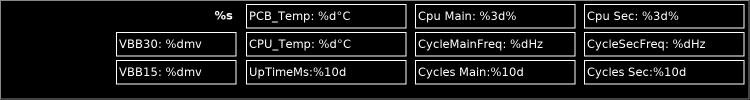
VISUALIZATION PLC_Status_Info  // 750x100
VAR_IN_OUT
	PlcStatus: SLL_IFM_CRXXXX.IFM_CRXXXX_System_STRUCT;
	Node: NodeComFB;
END_VAR
    Rectangle (246,32 160x24), "CPU_Temp: %d°C", text variable: PlcStatus.CPU_Temp
    Rectangle (415,60 160x24), "Cycles Main:%10d", text variable: PlcStatus.CycleCounter
    Rectangle (415,32 160x24), "CycleMainFreq: %dHz", text variable: PlcStatus.CycleFreq
    Rectangle (246,4 160x24), "PCB_Temp: %d°C", text variable: PlcStatus.PCB_Temp
    Rectangle (246,60 160x24), "UpTimeMs:%10d", text variable: PlcStatus.UpTimeMs
    Rectangle (116,32 120x24), "VBB30: %dmv", text variable: PlcStatus.VBB30_mV
    Rectangle (116,60 120x24), "VBB15: %dmv", text variable: PlcStatus.VBB15_mV
    Rectangle (71,4 165x23), "%s", text variable: Node.Full_Name
    Rectangle (584,4 160x24), "Cpu Sec: %3d%", text variable: TO_INT(PlcStatus.TaskInfo.fSecTaskCpuLoad)
    Rectangle (415,4 160x24), "Cpu Main: %3d%", text variable: TO_INT(PlcStatus.TaskInfo.fMainTaskCpuLoad)
    Rectangle (584,60 160x24), "Cycles Sec:%10d", text variable: PlcStatus.CycleSecCounter
    Rectangle (584,32 160x24), "CycleSecFreq: %dHz", text variable: PlcStatus.CycleSecFreq
END_VISUALIZATION

// Device/Application/LIBS/IO Diagnostics/IO Page Templates/PLC_Version_Info/PLC_Version_Info
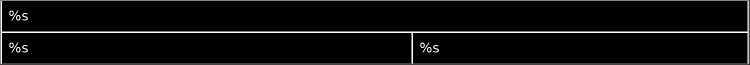
VISUALIZATION PLC_Version_Info  // 750x65
VAR_IN_OUT
	PlcVersion: PLC_Version_Unpack_FB;
END_VAR
    Textfield (1,0 747x32), "%s", text variable: PlcVersion.oMachine
    Textfield (1,32 411x32), "%s", text variable: PlcVersion.oVersion
    Textfield (412,32 336x32), "%s", text variable: PlcVersion.oCompiler
END_VISUALIZATION

// Device/Application/LIBS/IO Diagnostics/IO Page Objects/Output_Force
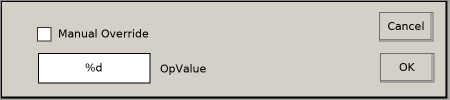
VISUALIZATION Output_Force  // 450x100
VAR_IN_OUT
	pOutputState: CRXXXX_OUTPUT_STATE_DATA;		
END_VAR
VAR
	flags: DWORD;
END_VAR
    Rectangle (0,0 447x98)
    Button (379,12 54x29), "Cancel"
        OnMouseClick:  Dialog=Current Dialog, Result=Cancel, NumpadKeypadSet=True
        OnMouseClick: execute { pOutputState.xManAuto:=0; }
    Button (380,53 54x29), "OK"
        OnMouseClick:  Dialog=Current Dialog, Result=OK, NumpadKeypadSet=True
    Checkbox (35,19 131x30), "Manual Override", variable: pOutputState.xManAuto
    Label (157,54 56x30), "OpValue"
    Rectangle (38,53 112x30), "%d", text variable: pOutputState.uiManValue
        OnMouseClick: write the text variable via VisuDialogs_Template.Numpad, min 0, max 5000, title 'Manual Value'
END_VISUALIZATION

// Device/Application/LIBS/IO Diagnostics/IO Page Objects/Output_IFM_PLC_CRXXXX_TITLE
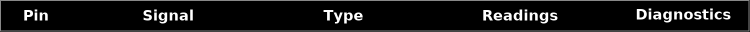
VISUALIZATION Output_IFM_PLC_CRXXXX_TITLE  // 750x32
    Textfield (398,3 244x25), "Readings"
    Textfield (629,2 109x25), "Diagnostics"
    Textfield (85,3 167x25), "Signal"
    Textfield (1,3 70x25), "Pin"
    Textfield (317,3 53x25), "Type"
END_VISUALIZATION

// Device/Application/LIBS/IO Diagnostics/IO Page Objects/Output_IFM_PLC_CRXXXX
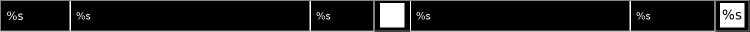
VISUALIZATION Output_IFM_PLC_CRXXXX  // 750x32
VAR_IN_OUT
	Output: CRXXXX_Output_Display;
END_VAR
VAR
END_VAR
    Textfield (410,0 220x32), "%s", text variable: Output.oMainString
        p55702900: Output.oMainStringColour
    Textfield (630,0 85x32), "%s", text variable: Output.oDiagStr
        p55702900: Output.oMainStringColour
    Textfield (70,0 240x32), "%s", text variable: Output.oSignalNameStr
    Textfield (0,0 70x32), "%s", text variable: Output.oPinDetailsStr
    Rectangle (380,3 24x24), invisible if: NOT Output.oShowDigRect, colour variable: Output.oDigRectColour
        p3450524324: Output.oDigRectColour
    Textfield (310,0 64x32), "%s", text variable: Output.oTypeStr
    Rectangle (720,3 24x24), "%s", text variable: Output.oForceText, invisible if: HMI_IO.Outputs_EnableAutoMan=0 OR Output.DisableMan=1, input disabled if: NOT HMI_IO.Outputs_EnableAutoMan OR GVL_System.HMI_OP_FORCE_DISABLE, colour variable: Output.oForceColour
        p3450524324: Output.oForceColour
        OnMouseClick:  Dialog=Output_Force, Parameters={flags: , pOutputState: Output.OpREF.OUTPUT_STATE_DATA}, Selected={1: , 0: }, OpenModal=True, OpenCentered=True
END_VISUALIZATION

// Device/Application/LIBS/IO Diagnostics/IO Page Objects/Input_IFM_PLC_CRXXXX
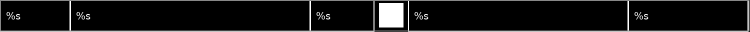
VISUALIZATION Input_IFM_PLC_CRXXXX  // 750x32
VAR_IN_OUT
	Input: CRXXXX_Input_Display;
END_VAR
VAR
END_VAR
    Textfield (408,0 220x32), "%s", text variable: Input.oMainString
        p55702900: Input.oMainStringColour
    Textfield (628,0 120x32), "%s", text variable: Input.oDiagStr
        p55702900: Input.oMainStringColour
    Textfield (70,0 240x32), "%s", text variable: Input.oSignalNameStr
    Textfield (0,0 70x32), "%s", text variable: Input.oPinDetailsStr
    Rectangle (379,3 24x24), invisible if: NOT Input.oShowDigRect, colour variable: Input.oDigRectColour
        p3450524324: Input.oDigRectColour
    Textfield (310,0 64x32), "%s", text variable: Input.oTypeStr
END_VISUALIZATION

// Device/Application/LIBS/IO Diagnostics/IO Page Objects/Input_IFM_PLC_CRXXXX_TITLE
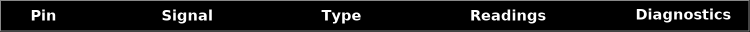
VISUALIZATION Input_IFM_PLC_CRXXXX_TITLE  // 750x32
    Textfield (386,3 244x25), "Readings"
    Textfield (629,2 109x25), "Diagnostics"
    Textfield (104,3 167x25), "Signal"
    Textfield (-1,3 89x25), "Pin"
    Textfield (315,3 53x25), "Type"
END_VISUALIZATION

// Device/Application/LIBS/IO Diagnostics/IO Page Objects/Output_Group_IFM_PLC_CRXXXX
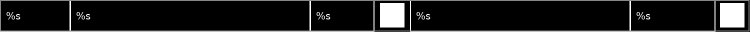
VISUALIZATION Output_Group_IFM_PLC_CRXXXX  // 750x32
{attribute 'VAR_IN_OUT_AS_POINTER'}
VAR_IN_OUT
	Output: CRXXXX_Output_Group_Display;
END_VAR
VAR
END_VAR
    Textfield (410,0 220x32), "%s", text variable: Output.oMainString
        p55702900: Output.oMainStringColour
    Textfield (630,0 85x32), "%s", text variable: Output.oDiagStr
        p55702900: Output.oMainStringColour
    Textfield (70,0 240x32), "%s", text variable: Output.oSignalNameStr
    Textfield (0,0 70x32), "%s", text variable: Output.oPinDetailsStr
    Rectangle (380,3 24x24), invisible if: NOT Output.oShowDigRect, colour variable: Output.oDigRectColour
        p3450524324: Output.oDigRectColour
    Textfield (310,0 64x32), "%s", text variable: Output.oTypeStr
    Rectangle (720,3 24x24), invisible if: NOT HMI_IO.Outputs_EnableAutoMan, input disabled if: NOT HMI_IO.Outputs_EnableAutoMan OR GVL_System.HMI_OP_FORCE_DISABLE
        OnMouseClick:  Dialog=Output_Force, Parameters={flags: , pOutputState: Output.OpGrpREF.OUTPUT_STATE_DATA}, Selected={1: , 0: }, OpenModal=True, OpenCentered=True
END_VISUALIZATION

// Device/Application/LIBS/IO Diagnostics/IO Page Templates/CR0709/Visualization_CR0709_Op_G0
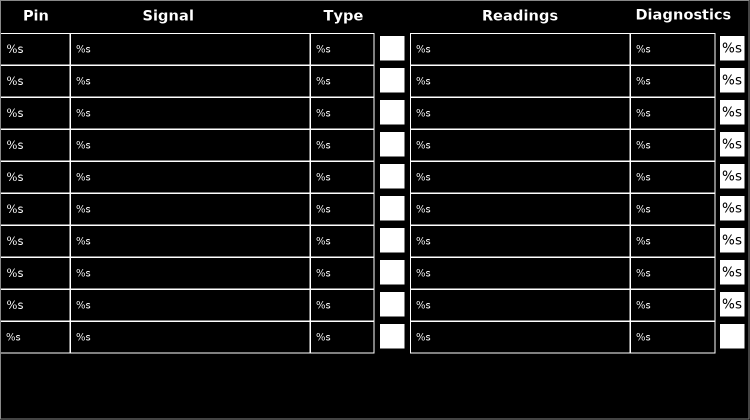
VISUALIZATION Visualization_CR0709_Op_G0  // 750x420
VAR_IN_OUT
	HMI_PLC_IO: HMI_PLC_CR0709_IO;
END_VAR
    Frame (0,33 800x32)
        shows Output_IFM_PLC_CRXXXX(Output := HMI_PLC_IO.OUT0000)
    Frame (0,0 800x32)
        shows Output_IFM_PLC_CRXXXX_TITLE()
    Frame (0,65 762x32)
        shows Output_IFM_PLC_CRXXXX(Output := HMI_PLC_IO.OUT0001)
    Frame (0,97 762x32)
        shows Output_IFM_PLC_CRXXXX(Output := HMI_PLC_IO.OUT0002)
    Frame (0,129 762x32)
        shows Output_IFM_PLC_CRXXXX(Output := HMI_PLC_IO.OUT0003)
    Frame (0,161 762x32)
        shows Output_IFM_PLC_CRXXXX(Output := HMI_PLC_IO.OUT0004)
    Frame (0,193 762x32)
        shows Output_IFM_PLC_CRXXXX(Output := HMI_PLC_IO.OUT0005)
    Frame (0,225 762x32)
        shows Output_IFM_PLC_CRXXXX(Output := HMI_PLC_IO.OUT0006)
    Frame (0,257 762x32)
        shows Output_IFM_PLC_CRXXXX(Output := HMI_PLC_IO.OUT0007)
    Frame (0,289 762x32)
        shows Output_IFM_PLC_CRXXXX(Output := HMI_PLC_IO.OUT0008)
    Frame (0,321 780x32)
        shows Output_Group_IFM_PLC_CRXXXX(Output := HMI_PLC_IO.GROUP0)
END_VISUALIZATION

// Device/Application/LIBS/IO Diagnostics/IO Page Templates/CR0709/Visualization_CR0709_Op_G2
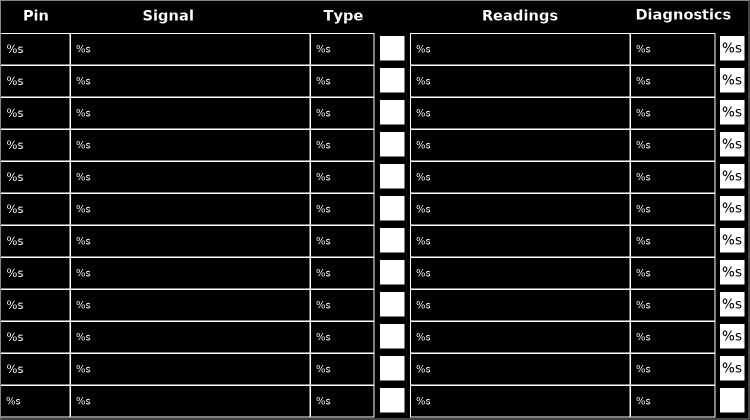
VISUALIZATION Visualization_CR0709_Op_G2  // 750x420
VAR_IN_OUT
	HMI_PLC_IO: HMI_PLC_CR0709_IO;
END_VAR
    Frame (0,33 762x32)
        shows Output_IFM_PLC_CRXXXX(Output := HMI_PLC_IO.OUT0200)
    Frame (0,0 800x32)
        shows Output_IFM_PLC_CRXXXX_TITLE()
    Frame (0,65 762x32)
        shows Output_IFM_PLC_CRXXXX(Output := HMI_PLC_IO.OUT0201)
    Frame (0,97 762x32)
        shows Output_IFM_PLC_CRXXXX(Output := HMI_PLC_IO.OUT0202)
    Frame (0,129 762x32)
        shows Output_IFM_PLC_CRXXXX(Output := HMI_PLC_IO.OUT0203)
    Frame (0,161 762x32)
        shows Output_IFM_PLC_CRXXXX(Output := HMI_PLC_IO.OUT0204)
    Frame (0,193 762x32)
        shows Output_IFM_PLC_CRXXXX(Output := HMI_PLC_IO.OUT0205)
    Frame (0,225 762x32)
        shows Output_IFM_PLC_CRXXXX(Output := HMI_PLC_IO.OUT0206)
    Frame (0,257 762x32)
        shows Output_IFM_PLC_CRXXXX(Output := HMI_PLC_IO.OUT0207)
    Frame (0,289 762x32)
        shows Output_IFM_PLC_CRXXXX(Output := HMI_PLC_IO.OUT0208)
    Frame (0,385 780x32)
        shows Output_Group_IFM_PLC_CRXXXX(Output := HMI_PLC_IO.GROUP2)
    Frame (0,321 762x32)
        shows Output_IFM_PLC_CRXXXX(Output := HMI_PLC_IO.OUT3000)
    Frame (0,353 762x32)
        shows Output_IFM_PLC_CRXXXX(Output := HMI_PLC_IO.OUT3001)
END_VISUALIZATION

// Device/Application/App_Common/Vizualisations/Main/Visualization_Net_Status_Adv
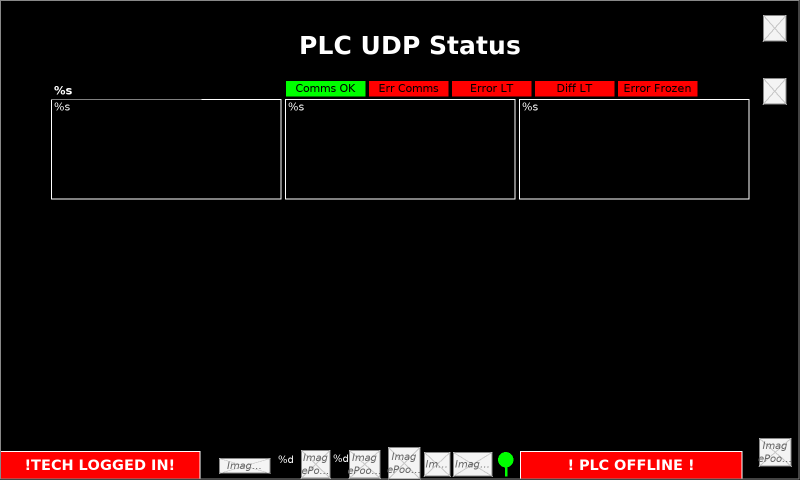
VISUALIZATION Visualization_Net_Status_Adv  // 800x480
    Frame (0,0 800x480)
        shows Visualization_Template()
    Label (219,30 382x30), "PLC UDP Status"
    Frame (50,80 700x120)
        shows PLC_UDP_Info(UDP_Info := PLC_SYSTEM.CHASSIS_UDP_Info_Viz)
    Image (763,15 23x26), invisible if: Nav.Footer_ShowNavLeft=0, image: ImagePool.Page_nav_left
    Image (763,78 23x26), invisible if: Nav.Footer_ShowNavRight=0, image: ImagePool.Page_nav_right
END_VISUALIZATION

// Device/Application/App_Common/Vizualisations/Main/Layout/Simulation/Visualization_SIM_IO
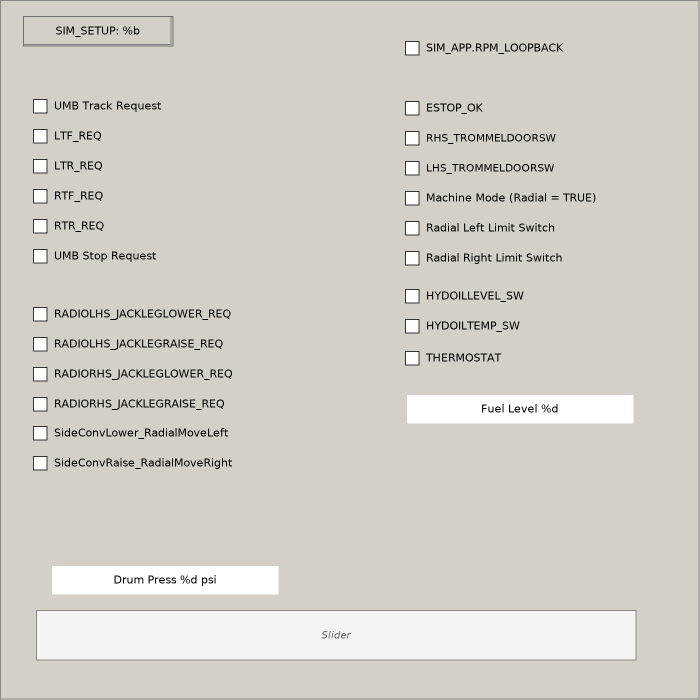
VISUALIZATION Visualization_SIM_IO  // 700x700
    Checkbox (403,33 188x30), "SIM_APP.RPM_LOOPBACK", variable: SIM_APP.RPM_LOOPBACK
    Checkbox (403,93 150x30), "ESTOP_OK", variable: Machine_IO.Inputs.ESTOP_OK.Dig
    Checkbox (403,123 150x30), "RHS_TROMMELDOORSW", variable: Machine_IO.Inputs.RHS_TROMMELDOORSW.Dig
    Checkbox (403,153 150x30), "LHS_TROMMELDOORSW", variable: Machine_IO.Inputs.LHS_TROMMELDOORSW.Dig
    Button (23,16 150x30), "SIM_SETUP: %b", text variable: SIM_APP.SIM_SETUP
        tap SIM_APP.SIM_SETUP
    Checkbox (403,183 231x30), "Machine Mode (Radial = TRUE)", variable: Machine_IO.Inputs.MachineMode.Dig
    Checkbox (403,213 250x30), "Radial Left Limit Switch", variable: Machine_IO.Inputs.Radial_LeftLimitSwitch.Dig
    Checkbox (403,243 250x30), "Radial Right Limit Switch", variable: Machine_IO.Inputs.Radial_RightLimitSwitch.Dig
    Checkbox (31,91 200x30), "UMB Track Request", variable: Machine_IO.Inputs.UMBTRACKREQ.Dig
    Checkbox (31,121 200x30), "LTF_REQ", variable: Machine_IO.Inputs.LTF_REQ.Dig
    Checkbox (31,151 200x30), "LTR_REQ", variable: Machine_IO.Inputs.LTR_REQ.Dig
    Checkbox (31,181 200x30), "RTF_REQ", variable: Machine_IO.Inputs.RTF_REQ.Dig
    Checkbox (31,211 200x30), "RTR_REQ", variable: Machine_IO.Inputs.RTR_REQ.Dig
    Checkbox (31,241 200x30), "UMB Stop Request", variable: Machine_IO.Inputs.UMBMACHINESTOP.Dig
    Slider (36,610 600x50), variable: Machine_IO.Inputs.DRUM_PRESSURE.ScaledReal, scale 0..3500
    Textfield (51,565 228x30), "Drum Press %d psi", text variable: Machine_IO.Inputs.DRUM_PRESSURE.ScaledReal
        OnMouseClick: write the text variable via Edit
    Checkbox (31,299 250x30), "RADIOLHS_JACKLEGLOWER_REQ", variable: Machine_IO.Inputs.RADIOLHS_JACKLEGLOWER_REQ.Dig
    Checkbox (31,329 250x30), "RADIOLHS_JACKLEGRAISE_REQ", variable: Machine_IO.Inputs.RADIOLHS_JACKLEGRAISE_REQ.Dig
    Checkbox (31,359 250x30), "RADIORHS_JACKLEGLOWER_REQ", variable: Machine_IO.Inputs.RADIORHS_JACKLEGLOWER_REQ.Dig
    Checkbox (31,389 250x30), "RADIORHS_JACKLEGRAISE_REQ", variable: Machine_IO.Inputs.RADIORHS_JACKLEGRAISE_REQ.Dig
    Checkbox (31,418 250x30), "SideConvLower_RadialMoveLeft", variable: Machine_IO.Inputs.SideConvLower_RadialMoveLeft.Dig
    Checkbox (31,448 250x30), "SideConvRaise_RadialMoveRight", variable: Machine_IO.Inputs.SideConvRaise_RadialMoveRight.Dig
    Checkbox (403,281 250x30), "HYDOILLEVEL_SW", variable: Machine_IO.Inputs.HYDOILLEVEL_SW.Dig
    Checkbox (403,311 250x30), "HYDOILTEMP_SW", variable: Machine_IO.Inputs.HYDOILTEMP_SW.Dig
    Checkbox (403,343 250x30), "THERMOSTAT", variable: Machine_IO.Inputs.THERMOSTAT.Dig
    Textfield (406,394 228x30), "Fuel Level %d", text variable: Machine_IO.Inputs.FUELLEVEL_PERCENT.ScaledReal
        OnMouseClick: write the text variable via Edit
END_VISUALIZATION

// Device/Application/App_Common/Vizualisations/Main/Visualization_Net_Status
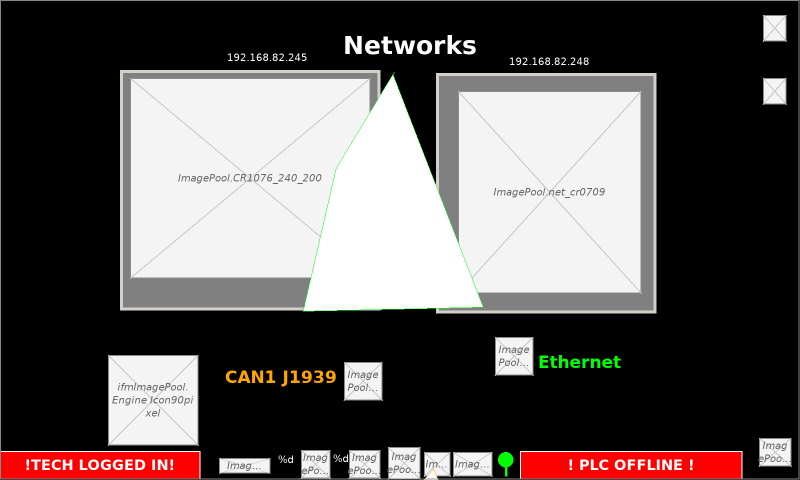
VISUALIZATION Visualization_Net_Status  // 800x480
    Frame (0,0 800x480)
        shows Visualization_Template()
    Frame (0,21 800x424)
        shows Visualization_Net_Background()
    Polygon (483,307) (303,311) (336,168) (394,72) (393,75)
    Label (190,363 150x28), "CAN1 J1939"
    Label (535,348 174x28), "Ethernet"
    Label (219,30 382x30), "Networks"
    Polygon (507,639) (389,729) (311,591) (433,470) (433,468)
    Image (495,337 38x38), invisible if: UDP_COMS_RX.CHASSIS_PLC_RED_CROSS=0, image: ImagePool.red-cross
    Image (344,362 38x38), invisible if: GVL_Engine.EngineHrs>0, image: ImagePool.red-cross
    Image (763,15 23x26), invisible if: Nav.Footer_ShowNavLeft=0, image: ImagePool.Page_nav_left
    Image (763,78 23x26), invisible if: Nav.Footer_ShowNavRight=0, image: ImagePool.Page_nav_right
    Image (108,355 90x90), image: ifmImagePool.Engine Icon90pixel
END_VISUALIZATION

// Device/Application/LIBS/IO Diagnostics/IO Page Templates/CR0709/Visualization_CR0709_Ip_G0
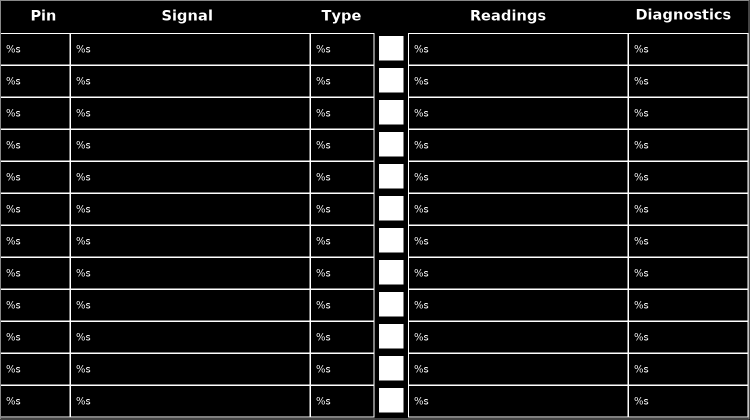
VISUALIZATION Visualization_CR0709_Ip_G0  // 750x420
VAR_IN_OUT
	HMI_PLC_IO: HMI_PLC_CR0709_IO;
END_VAR
    Frame (0,33 762x32)
        shows Input_IFM_PLC_CRXXXX(Input := HMI_PLC_IO.IN0100)
    Frame (0,0 750x32)
        shows Input_IFM_PLC_CRXXXX_TITLE()
    Frame (0,65 762x32)
        shows Input_IFM_PLC_CRXXXX(Input := HMI_PLC_IO.IN0101)
    Frame (0,97 762x32)
        shows Input_IFM_PLC_CRXXXX(Input := HMI_PLC_IO.IN0102)
    Frame (0,129 762x32)
        shows Input_IFM_PLC_CRXXXX(Input := HMI_PLC_IO.IN0103)
    Frame (0,161 762x32)
        shows Input_IFM_PLC_CRXXXX(Input := HMI_PLC_IO.IN0200)
    Frame (0,193 762x32)
        shows Input_IFM_PLC_CRXXXX(Input := HMI_PLC_IO.IN0201)
    Frame (0,225 762x32)
        shows Input_IFM_PLC_CRXXXX(Input := HMI_PLC_IO.IN0202)
    Frame (0,257 762x32)
        shows Input_IFM_PLC_CRXXXX(Input := HMI_PLC_IO.IN0203)
    Frame (0,289 762x32)
        shows Input_IFM_PLC_CRXXXX(Input := HMI_PLC_IO.IN0600)
    Frame (0,321 762x32)
        shows Input_IFM_PLC_CRXXXX(Input := HMI_PLC_IO.IN0601)
    Frame (0,353 762x32)
        shows Input_IFM_PLC_CRXXXX(Input := HMI_PLC_IO.IN0602)
    Frame (0,385 762x32)
        shows Input_IFM_PLC_CRXXXX(Input := HMI_PLC_IO.IN0603)
END_VISUALIZATION

// Device/Application/LIBS/IO Diagnostics/IO Page Templates/CR0709/Visualization_CR0709_Ip_G1
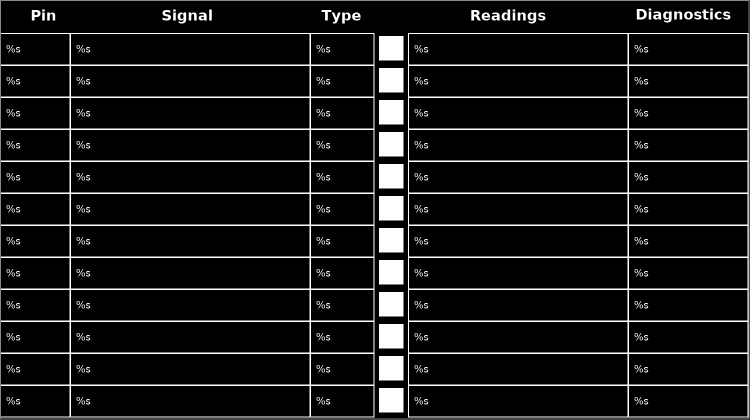
VISUALIZATION Visualization_CR0709_Ip_G1  // 750x420
VAR_IN_OUT
	HMI_PLC_IO: HMI_PLC_CR0709_IO;
END_VAR
    Frame (0,33 762x32)
        shows Input_IFM_PLC_CRXXXX(Input := HMI_PLC_IO.IN0700)
    Frame (0,0 801x32)
        shows Input_IFM_PLC_CRXXXX_TITLE()
    Frame (0,65 762x32)
        shows Input_IFM_PLC_CRXXXX(Input := HMI_PLC_IO.IN0701)
    Frame (0,97 762x32)
        shows Input_IFM_PLC_CRXXXX(Input := HMI_PLC_IO.IN0702)
    Frame (0,129 762x32)
        shows Input_IFM_PLC_CRXXXX(Input := HMI_PLC_IO.IN0703)
    Frame (0,161 762x32)
        shows Input_IFM_PLC_CRXXXX(Input := HMI_PLC_IO.IN0000)
    Frame (0,193 762x32)
        shows Input_IFM_PLC_CRXXXX(Input := HMI_PLC_IO.IN0001)
    Frame (0,225 762x32)
        shows Input_IFM_PLC_CRXXXX(Input := HMI_PLC_IO.IN0002)
    Frame (0,257 762x32)
        shows Input_IFM_PLC_CRXXXX(Input := HMI_PLC_IO.IN0003)
    Frame (0,289 762x32)
        shows Input_IFM_PLC_CRXXXX(Input := HMI_PLC_IO.IN0500)
    Frame (0,321 762x32)
        shows Input_IFM_PLC_CRXXXX(Input := HMI_PLC_IO.IN0501)
    Frame (0,353 762x32)
        shows Input_IFM_PLC_CRXXXX(Input := HMI_PLC_IO.IN0502)
    Frame (0,385 762x32)
        shows Input_IFM_PLC_CRXXXX(Input := HMI_PLC_IO.IN0503)
END_VISUALIZATION

// Device/Application/App_Common/Vizualisations/Main/Layout/Visualization_Net_Background
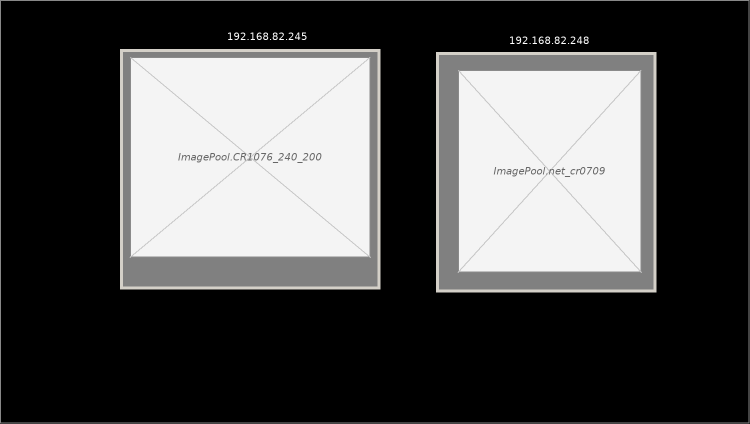
VISUALIZATION Visualization_Net_Background  // 750x424
    Rectangle (120,49 260x240)
    Rectangle (436,52 220x240)
    Image (458,70 183x202), image: ImagePool.net_cr0709
    Rectangle (501,31 97x19), "192.168.82.248"
    Rectangle (219,27 97x19), "192.168.82.245"
    Image (130,57 240x200), image: ImagePool.CR1076_240_200
END_VISUALIZATION

// Device/Application/App_Common/Vizualisations/Main/Visualization_Settings_Misc
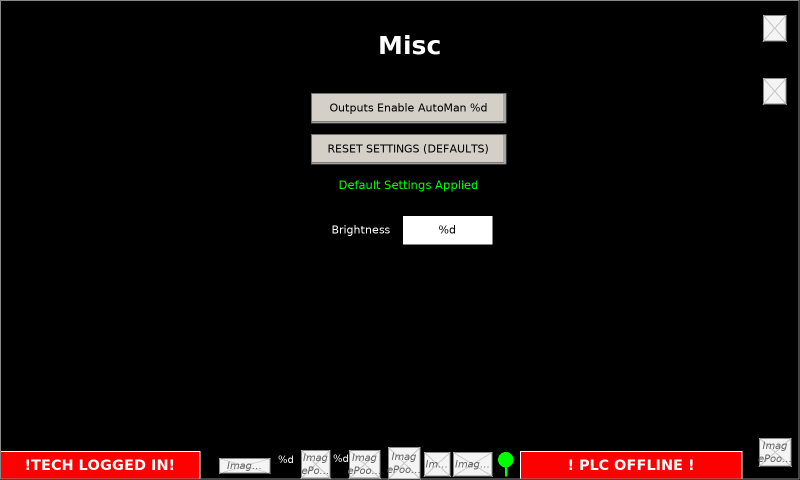
VISUALIZATION Visualization_Settings_Misc  // 800x480
    Frame (0,0 800x480)
        shows Visualization_Template()
    Label (219,30 382x30), "Misc"
    Button (311,93 195x30), "Outputs Enable AutoMan %d", text variable: HMI_IO.Outputs_EnableAutoMan, invisible if: NOT GVL_System.Access_Level_Tech
        toggle HMI_IO.Outputs_EnableAutoMan
    Label (317,215 76x30), "Brightness"
    Rectangle (402,215 91x30), "%d", text variable: GVL_Persistant.Brightness
        OnValueChanged: execute {  }
        OnValueChanged: write the text variable via Default, min LCD_Brighness_Control.Brightness_Min, max LCD_Brighness_Control.Brightness_Max
        OnMouseClick: write the text variable via VisuDialogs_Template.Numpad, min 10, max 100, title 'Brighntess %'
    Button (311,134 195x30), "RESET SETTINGS (DEFAULTS)", invisible if: GVL_System.Access_Level_Tech=0
        tap PLC_SYSTEM.Reset_Settings
    Label (311,174 195x22), "Default Settings Applied", invisible if: PLC_SYSTEM.Reset_Settings_Applied=0
    Image (763,15 23x26), invisible if: Nav.Footer_ShowNavLeft=0, image: ImagePool.Page_nav_left
    Image (763,78 23x26), invisible if: Nav.Footer_ShowNavRight=0, image: ImagePool.Page_nav_right
END_VISUALIZATION

// Device/Application/App_Common/Vizualisations/Main/Visualization_PLC_Status
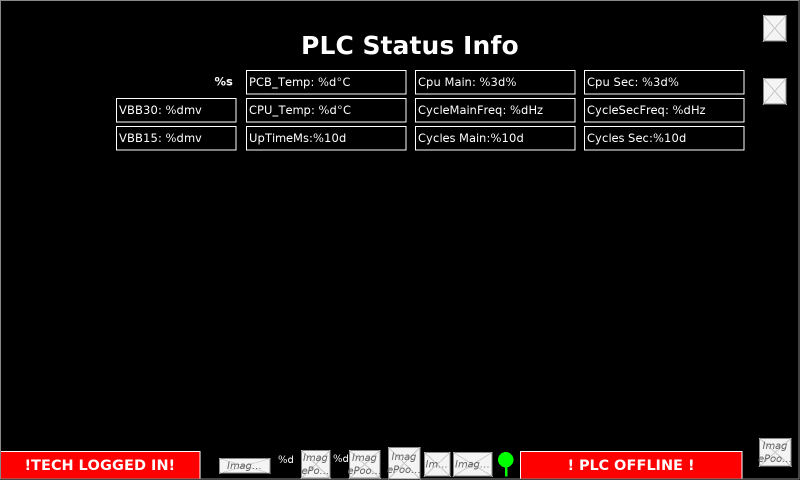
VISUALIZATION Visualization_PLC_Status  // 800x480
    Frame (0,0 800x480)
        shows Visualization_Template()
    Label (219,30 382x30), "PLC Status Info"
    Frame (0,66 800x65)
        shows PLC_Status_Info(PlcStatus := NVL_IO_CHASSIS.System, Node := Machine_IO.Node_CHASSIS)
    Image (763,15 23x26), invisible if: Nav.Footer_ShowNavLeft=0, image: ImagePool.Page_nav_left
    Image (763,78 23x26), invisible if: Nav.Footer_ShowNavRight=0, image: ImagePool.Page_nav_right
END_VISUALIZATION

// Device/Application/App_Common/Vizualisations/Main/Visualization_Settings_RTC
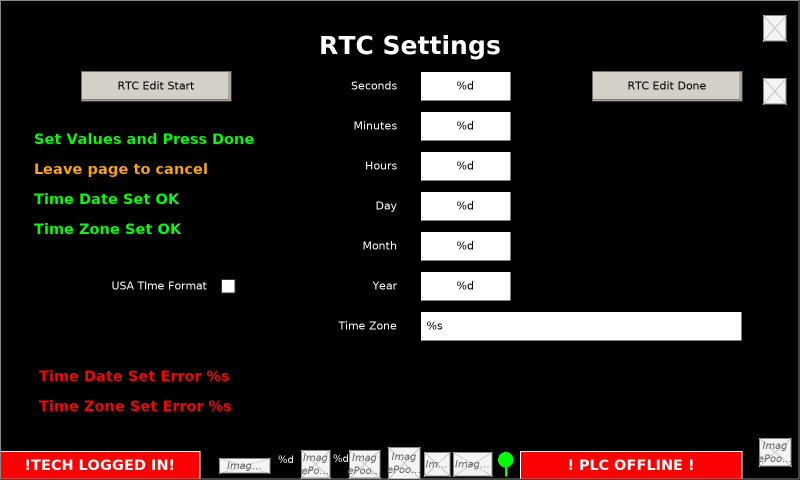
VISUALIZATION Visualization_Settings_RTC  // 800x480
    Frame (0,0 800x480)
        shows Visualization_Template()
    Label (219,30 382x30), "RTC Settings"
    Label (300,271 100x30), "Year"
    Rectangle (420,271 91x30), "%d", text variable: CR1140_RTC_Edit.RTC_Temp.uiYear, input disabled if: CR1140_RTC_Edit.RTC_Edit_Start=0
        OnValueChanged: execute { CR1140_RTC_Edit.RTC_Edit_Start:=1; }
        OnMouseClick: write the text variable via VisuDialogs_Template.Numpad, min 2000, max 3000, title 'Years in YYYYY format'
    Label (300,231 100x30), "Month"
    Rectangle (420,231 91x30), "%d", text variable: CR1140_RTC_Edit.RTC_Temp.uiMonth, input disabled if: CR1140_RTC_Edit.RTC_Edit_Start=0
        OnValueChanged: execute { CR1140_RTC_Edit.RTC_Edit_Start:=1; }
        OnMouseClick: write the text variable via VisuDialogs_Template.Numpad, min 1, max 12, title 'Month'
    Label (300,191 100x30), "Day"
    Rectangle (420,191 91x30), "%d", text variable: CR1140_RTC_Edit.RTC_Temp.uiDay, input disabled if: CR1140_RTC_Edit.RTC_Edit_Start=0
        OnValueChanged: execute { CR1140_RTC_Edit.RTC_Edit_Start:=1; }
        OnMouseClick: write the text variable via VisuDialogs_Template.Numpad, min 1, max 31, title 'Day of Month'
    Label (300,151 100x30), "Hours"
    Rectangle (420,151 91x30), "%d", text variable: CR1140_RTC_Edit.RTC_Temp.uiHour, input disabled if: CR1140_RTC_Edit.RTC_Edit_Start=0
        OnValueChanged: execute { CR1140_RTC_Edit.RTC_Edit_Start:=1; }
        OnMouseClick: write the text variable via VisuDialogs_Template.Numpad, min 0, max 23, title 'Hours (24hr)'
    Label (300,111 100x30), "Minutes"
    Rectangle (420,111 91x30), "%d", text variable: CR1140_RTC_Edit.RTC_Temp.uiMinute, input disabled if: CR1140_RTC_Edit.RTC_Edit_Start=0
        OnValueChanged: execute { CR1140_RTC_Edit.RTC_Edit_Start:=1; }
        OnMouseClick: write the text variable via VisuDialogs_Template.Numpad, min 0, max 59, title 'Minutes'
    Label (300,71 100x30), "Seconds"
    Rectangle (420,71 91x30), "%d", text variable: CR1140_RTC_Edit.RTC_Temp.uiSeconds, input disabled if: CR1140_RTC_Edit.RTC_Edit_Start=0
        OnValueChanged: execute { CR1140_RTC_Edit.RTC_Edit_Start:=1; }
        OnMouseClick: write the text variable via VisuDialogs_Template.Numpad, min 0, max 59, title 'Secondst'
    Button (81,71 150x30), "RTC Edit Start"
        toggle CR1140_RTC_Edit.RTC_Edit_Start p2164770859=TRUE
    Button (592,71 150x30), "RTC Edit Done", input disabled if: CR1140_RTC_Edit.RTC_Edit_Start=0
        tap CR1140_RTC_Edit.RTC_Edit_Done
    Label (31,124 250x30), "Set Values and Press Done", invisible if: CR1140_RTC_Edit.RTC_Edit_Start=0
    Label (31,154 250x30), "Leave page to cancel", invisible if: CR1140_RTC_Edit.RTC_Edit_Start=0
    Label (300,311 100x30), "Time Zone"
    Rectangle (420,311 322x30), "%s", text variable: CR1140_RTC_Edit.RTC_Timezone, input disabled if: CR1140_RTC_Edit.RTC_Edit_Start=0
        OnValueChanged: execute { CR1140_RTC_Edit.RTC_Edit_Start:=1; }
        OnMouseClick: write the text variable via VisuDialogs_Template.Keypad, title 'Time Zone - see docs'
    Label (31,184 250x30), "Time Date Set OK", invisible if: CR1140_RTC_Edit.TimeDateSetOK=0
    Label (31,214 250x30), "Time Zone Set OK", invisible if: CR1140_RTC_Edit.ZoneSetOK=0
    Rectangle (31,391 700x30), "Time Zone Set Error %s", text variable: CR1140_RTC_Edit.ZoneSetErrorCode, invisible if: CR1140_RTC_Edit.ZoneSetError=0
    Rectangle (31,361 700x30), "Time Date Set Error %s", text variable: CR1140_RTC_Edit.TimeDateSetErrorCode, invisible if: CR1140_RTC_Edit.TimeDateSetError=0
    Checkbox (219,271 33x30), variable: GVL_Persistant.Sys_Settings.USA_TIme_Format
    Label (94,271 116x30), "USA TIme Format"
    Image (763,15 23x26), invisible if: Nav.Footer_ShowNavLeft=0, image: ImagePool.Page_nav_left
    Image (763,78 23x26), invisible if: Nav.Footer_ShowNavRight=0, image: ImagePool.Page_nav_right
END_VISUALIZATION

// Device/Application/App_Common/Vizualisations/Main/Layout/Simulation/Visualization_SIM_IO_AUX
VISUALIZATION Visualization_SIM_IO_AUX  // 700x700
END_VISUALIZATION

// Device/Application/App_Common/Vizualisations/Main/Visualization_Settings_IO_Log
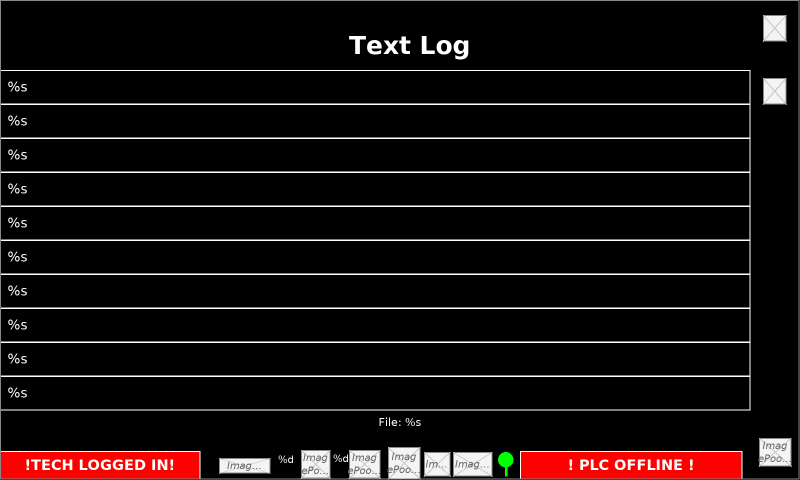
VISUALIZATION Visualization_Settings_IO_Log  // 800x480
    Frame (0,0 800x480)
        shows Visualization_Template()
    Label (219,30 382x30), "Text Log"
    Rectangle (0,70 750x34), "%s", text variable: PLC_LOGGING.LOG_LINES[0]
    Rectangle (0,104 750x34), "%s", text variable: PLC_LOGGING.LOG_LINES[1]
    Rectangle (0,138 750x34), "%s", text variable: PLC_LOGGING.LOG_LINES[2]
    Rectangle (0,172 750x34), "%s", text variable: PLC_LOGGING.LOG_LINES[3]
    Rectangle (0,206 750x34), "%s", text variable: PLC_LOGGING.LOG_LINES[4]
    Rectangle (0,240 750x34), "%s", text variable: PLC_LOGGING.LOG_LINES[5]
    Rectangle (0,274 750x34), "%s", text variable: PLC_LOGGING.LOG_LINES[6]
    Rectangle (0,308 750x34), "%s", text variable: PLC_LOGGING.LOG_LINES[7]
    Rectangle (0,342 750x34), "%s", text variable: PLC_LOGGING.LOG_LINES[8]
    Rectangle (0,376 750x34), "%s", text variable: PLC_LOGGING.LOG_LINES[9]
    Rectangle (250,410 300x25), "File: %s", text variable: GVL_Logging.Main_Log_Filename
    Image (763,15 23x26), invisible if: Nav.Footer_ShowNavLeft=0, image: ImagePool.Page_nav_left
    Image (763,78 23x26), invisible if: Nav.Footer_ShowNavRight=0, image: ImagePool.Page_nav_right
END_VISUALIZATION

// Device/Application/App_Common/Vizualisations/Main/Visualization_Settings_1
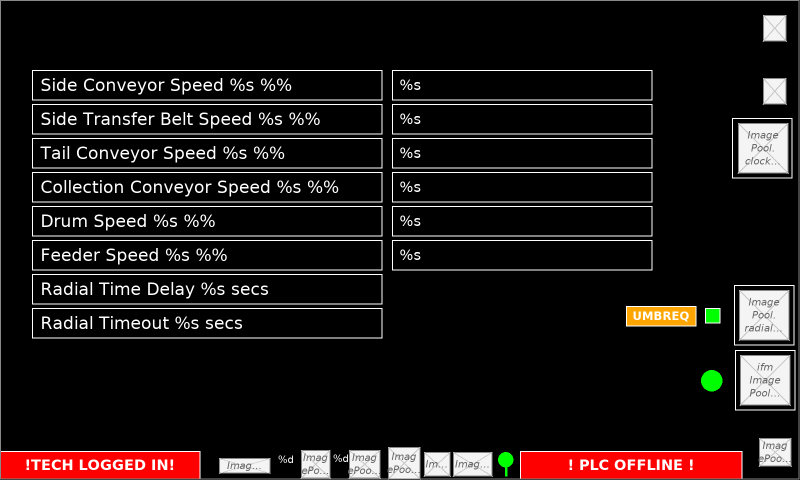
VISUALIZATION Visualization_Settings_1  // 800x480
    Frame (0,0 800x480)
        shows Visualization_Template()
    Rectangle (32,240 350x30), "Feeder Speed %s %%", text variable: GVL_Persistant.App_Settings.FeederSpd_Percent
        OnMouseClick: write the text variable via VisuDialogs_Template.Numpad, min 0, max 100, title "Feeder Speed %"
    Rectangle (32,206 350x30), "Drum Speed %s %%", text variable: GVL_Persistant.App_Settings.DrumSpd_Percent
        OnMouseClick: write the text variable via VisuDialogs_Template.Numpad, min 0, max 100, title "Drum Speed %"
    Rectangle (32,172 350x30), "Collection Conveyor Speed %s %%", text variable: GVL_Persistant.App_Settings.CollectConvSpd_Percent
        OnMouseClick: write the text variable via VisuDialogs_Template.Numpad, min 0, max 100, title "Collection Conveyor Speed %"
    Rectangle (32,70 350x30), "Stockpile Conv Speed %s %%", text variable: GVL_Persistant.App_Settings.SideConvSpd_Percent, invisible if: GVL_APP.MachineModelRadial=0
        OnMouseClick: write the text variable via VisuDialogs_Template.Numpad, min 0, max 100, title "Stockpile Conv. Speed %"
    Rectangle (32,138 350x30), "Tail Conveyor Speed %s %%", text variable: GVL_Persistant.App_Settings.TailConvSpd_Percent
        OnMouseClick: write the text variable via VisuDialogs_Template.Numpad, min 0, max 100, title "Tail Conveyor Speed %"
    Image (740,355 50x50), image: ifmImagePool.LeverValve50pixel
    Ellipse (701,370 21x21), invisible if: GVL_Machine.SetupDumpValveOn=0
    RoundedRectangle (735,350 60x60)
    Image (763,15 23x26), invisible if: Nav.Footer_ShowNavLeft=0, image: ImagePool.Page_nav_left
    Image (763,78 23x26), invisible if: Nav.Footer_ShowNavRight=0, image: ImagePool.Page_nav_right
    Rectangle (392,240 260x30), "%s", text variable: AutoManSelButtons.PWM_Op_FeederSpeed_Status_Str
        OnMouseClick: write the text variable via VisuDialogs_Template.Numpad, min 0, max 100, title "Feeder Speed %"
    Rectangle (392,206 260x30), "%s", text variable: AutoManSelButtons.PWM_Op_DrumSpeed_Status_Str
        OnMouseClick: write the text variable via VisuDialogs_Template.Numpad, min 0, max 100, title "Feeder Speed %"
    Rectangle (392,172 260x30), "%s", text variable: AutoManSelButtons.PWM_Op_CollectionConveyor_Status_Str
        OnMouseClick: write the text variable via VisuDialogs_Template.Numpad, min 0, max 100, title "Feeder Speed %"
    Rectangle (392,138 260x30), "%s", text variable: AutoManSelButtons.PWM_Op_TailConveyor_Status_Str
        OnMouseClick: write the text variable via VisuDialogs_Template.Numpad, min 0, max 100, title "Feeder Speed %"
    Rectangle (392,104 260x30), "%s", text variable: AutoManSelButtons.PWM_Op_SideTransfer_Status_Str, invisible if: GVL_APP.MachineModelRadial=1
        OnMouseClick: write the text variable via VisuDialogs_Template.Numpad, min 0, max 100, title "Feeder Speed %"
    Rectangle (392,70 260x30), "%s", text variable: AutoManSelButtons.PWM_Op_SideConveyor_Status_Str
        OnMouseClick: write the text variable via VisuDialogs_Template.Numpad, min 0, max 100, title "Feeder Speed %"
    Image (738,123 48x50), invisible if: GVL_APP.MachineModelRadial=0, image: ImagePool.swt_50_50
    RoundedRectangle (732,118 60x60), invisible if: GVL_APP.MachineModelRadial=0
    Image (738,123 50x50), invisible if: GVL_APP.AutoRadialTimed=0 OR GVL_APP.MachineModelRadial=0, image: ImagePool.clock_50_50
    RoundedRectangle (734,285 60x60), invisible if: GVL_APP.MachineModelRadial=0
    Image (739,290 50x50), invisible if: GVL_APP.MachineModelRadial=0, image: ImagePool.radial_50_50
    Rectangle (705,308 15x15), invisible if: GVL_APP.AutoRadialModeIcon=0 OR GVL_APP.MachineModelRadial=0
    Rectangle (32,274 350x30), "Radial Time Delay %s secs", text variable: GVL_Persistant.App_Settings.RadialTimeDelay_SP, invisible if: GVL_APP.MachineModelRadial=0
        OnMouseClick: write the text variable via VisuDialogs_Template.Numpad, min 30, max 300, title "Radial Time Delay"
    Rectangle (32,308 350x30), "Radial Timeout %s secs", text variable: GVL_Persistant.App_Settings.RadialTimeOut_SP, invisible if: GVL_APP.MachineModelRadial=0
        OnMouseClick: write the text variable via VisuDialogs_Template.Numpad, min 10, max 300, title "Radial Timeout"
    Rectangle (32,104 350x30), "Side Transfer Belt Speed %s %%", text variable: GVL_Persistant.App_Settings.SideTransferConvSpd_Percent, invisible if: GVL_APP.MachineModelRadial=1
        OnMouseClick: write the text variable via VisuDialogs_Template.Numpad, min 0, max 100, title "Side Transfer Belt Speed %"
    Rectangle (32,70 350x30), "Side Conveyor Speed %s %%", text variable: GVL_Persistant.App_Settings.SideConvSpd_Percent, invisible if: GVL_APP.MachineModelRadial=1
        OnMouseClick: write the text variable via VisuDialogs_Template.Numpad, min 0, max 100, title "Side Conveyor Speed %"
    RoundedRectangle (626,306 70x20), "UMBREQ", invisible if: Machine_IO.Inputs.UMBTRACKREQ.Dig=0 OR GVL_APP.MachineModelRadial=0
END_VISUALIZATION

// Device/Application/LIBS/Alarms/Viz/Alarm_Logger_Title
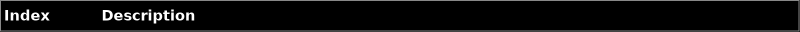
VISUALIZATION Alarm_Logger_Title  // 800x32
    Textfield (65,3 167x25), "Description"
    Textfield (1,3 89x25), "Index"
END_VISUALIZATION

// Device/Application/LIBS/Alarms/Viz/Alarm_Logger_Line
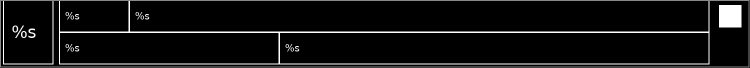
VISUALIZATION Alarm_Logger_Line  // 750x68
VAR_IN_OUT
	Item: Alarm_Logger_Line_FB;
END_VAR
VAR
END_VAR
    Textfield (279,32 430x32), "%s", text variable: Item.oAdd_Info
    Textfield (129,0 580x32), "%s", text variable: Item.oDescription
    Textfield (3,0 50x64), "%s", text variable: Item.oIndex
    Textfield (59,32 220x32), "%s", text variable: Item.oTime
    Rectangle (718,4 24x24), colour variable: Item.oSquareColour
    Textfield (59,0 70x32), "%s", text variable: Item.oID
END_VISUALIZATION

// Device/Application/LIBS/Alarms/Viz/Alarm_Logger_Table
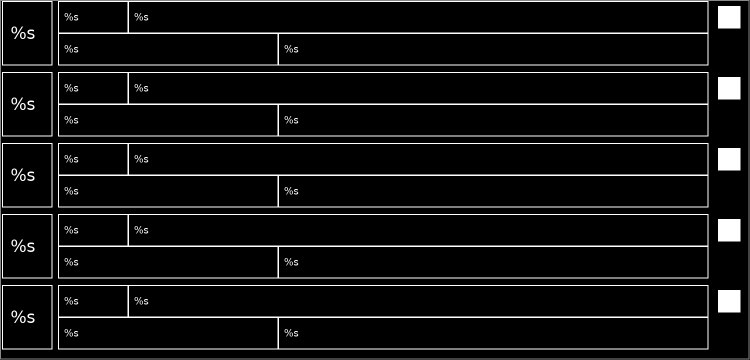
VISUALIZATION Alarm_Logger_Table  // 750x360
VAR_IN_OUT
	LINE: ARRAY [0..4] OF Alarm_Logger_Line_FB;
END_VAR
    Frame (-1,1 800x32)
        shows Alarm_Logger_Line(Item := LINE[0])
    Frame (-1,72 800x32)
        shows Alarm_Logger_Line(Item := LINE[1])
    Frame (-1,143 800x32)
        shows Alarm_Logger_Line(Item := LINE[2])
    Frame (-1,214 800x32)
        shows Alarm_Logger_Line(Item := LINE[3])
    Frame (-1,285 800x32)
        shows Alarm_Logger_Line(Item := LINE[4])
END_VISUALIZATION

// Device/Application/App_Common/Vizualisations/Main/Visualization_Main_1
